// TIA Portal V20 export
DATA_BLOCK "PM10"   // DB284
// stored: MemoryReserve 100
   VAR
      "STACK NG CLAMP MOVER CLOSE" : Bool;
      "STACK NG CLAMP MOVER OPEN" : Bool;
      "STACK NG CLAMP LEFT CLOSE" : Bool;
      "STACK NG CLAMP LEFT OPEN" : Bool;
      "STACK NG CLAMP RIGHT CLOSE" : Bool;
      "STACK NG CLAMP RIGHT OPEN" : Bool;
      "STACK NG CLAMP Z-AXIS UP" : Bool;
      "STACK NG CLAMP Z-AXIS DOWN" : Bool;
      "STACK NG CLAMP MOVER FORWARD" : Bool;
      "STACK NG CLAMP MOVER BACKWARD" : Bool;
      "STACK NG BOX LIFT UP" : Bool;
      "STACK NG BOX LIFT DOWN" : Bool;
      "STACK NG BOX LOCK UP" : Bool;
      "STACK NG BOX LOCK DOWN" : Bool;
      SPARE : Bool;
      SPARE_1 : Bool;
   END_VAR
BEGIN
END_DATA_BLOCK
